INTERFACE ITmsMover EXTENDS IMover

METHOD ActivateTrack : BOOL
VAR_INPUT
	newTrack : OTCID;
END_VAR
END_METHOD

PROPERTY ActiveTrack : OTCID
GET
END_GET
END_PROPERTY

METHOD SetMoverInterface : BOOL
VAR_INPUT
	MoverInterface : I_TcIoXtsXpuMover;
END_VAR
END_METHOD

END_INTERFACE

(* stored: Version 1.1.0.1, ProductVersion 3.1.4024.12
   Itf ITmsMover: Id {1dd4f0e1-1fa2-4d8b-bd4e-d91c7c33d591}
   Method ActivateTrack: Id {6e62ed33-5211-41f4-b2cf-01546af65477}
   Property ActiveTrack: Id {c110d4d3-e578-42cb-b306-1d0f5bc49fd5}
   Get Get: Id {1c67a4ef-4755-4dc5-b029-4a5b040fcdbc}
   Method SetMoverInterface: Id {b12088fd-1d05-4423-b53f-cb9b8228c3e3} *)
